FUNCTION_BLOCK ABSTRACT FB_ESSMonitoringBase
VAR_INPUT
    nEcMasterNetId: T_AmsNetId;
    iSafetyProvider: I_SafetyProvider;
END_VAR
VAR_OUTPUT
    aErrorID: ARRAY [1..nMAX_ALARMS] OF INT;
    aErrorMsg: ARRAY [1..nMAX_ALARMS] OF STRING;
    nEcMasterFramesLost: UDINT;
    nCPULoad: UDINT;
    fCycleExecTime_ms: REAL;
    nAlarmGrpBitNumber: UDINT;
END_VAR
VAR
    _bErrorAcknowledgeButton: BOOL;
    _bErrorAcknowledgeLED: BOOL;
    _bStatusLED: BOOL;
    _bEStopLED: BOOL;
    _bErrorLED: BOOL;
    _bEStopReleased: BOOL;
    _nEcMasterDevState: UINT;

    aAlarmList: ARRAY [1..nMAX_ALARMS] OF ST_MonitoringAlarm := [
(*[1]*)(nErrorID:=241, sErrorMsg:='The DC OK Status from PS 24V-1 is OFF.', eStatusLED:=E_MonitorLed.eFast, eErrorLED:=E_MonitorLed.eSteady),
(*[2]*)(nErrorID:=242, sErrorMsg:='The DC OK Status from PS 24V-2 is OFF.', eStatusLED:=E_MonitorLed.eFast, eErrorLED:=E_MonitorLed.eSteady),
(*[3]*)(nErrorID:=243, sErrorMsg:='The DC OK Status from PS 24V-3 is OFF.', eStatusLED:=E_MonitorLed.eFast, eErrorLED:=E_MonitorLed.eSteady),
(*[4]*)(nErrorID:=481, sErrorMsg:='The DC OK Status from PS 48V-1 is OFF.', eStatusLED:=E_MonitorLed.eFast, eErrorLED:=E_MonitorLed.eSteady),
(*[5]*)(nErrorID:=482, sErrorMsg:='The DC OK Status from PS 48V-2 is OFF.', eStatusLED:=E_MonitorLed.eFast, eErrorLED:=E_MonitorLed.eSteady),
(*[6]*)(nErrorID:=483, sErrorMsg:='The DC OK Status from PS 48V-3 is OFF.', eStatusLED:=E_MonitorLed.eFast, eErrorLED:=E_MonitorLed.eSteady),
(*[7]*)(nErrorID:=484, sErrorMsg:='The DC OK Status from PS 48V-4 is OFF.', eStatusLED:=E_MonitorLed.eFast, eErrorLED:=E_MonitorLed.eSteady),
(*[8]*)(nErrorID:=11, sErrorMsg:='MCB Fan OK status is OFF', eStatusLED:=E_MonitorLed.eFast, eErrorLED:=E_MonitorLed.eSteady),
(*[9]*)(nErrorID:=12, sErrorMsg:='SPD OK status is OFF', eStatusLED:=E_MonitorLed.eFast, eErrorLED:=E_MonitorLed.eSteady),
(*[10]*)(nErrorID:=13, sErrorMsg:='Cabinet door Opened', eStatusLED:=E_MonitorLed.eSteady, eErrorLED:=E_MonitorLed.eSteady, bLedAutoReset:=TRUE),
(*[11]*)(nErrorID:=301, sErrorMsg:='Fuse 1 tripped', eStatusLED:=E_MonitorLed.eUndefined, eErrorLED:=E_MonitorLed.eUndefined),
(*[12]*)(nErrorID:=302, sErrorMsg:='Fuse 2 tripped', eStatusLED:=E_MonitorLed.eSlow, eErrorLED:=E_MonitorLed.eSteady),
(*[13]*)(nErrorID:=303, sErrorMsg:='Fuse 3 tripped', eStatusLED:=E_MonitorLed.eSlow, eErrorLED:=E_MonitorLed.eSteady),
(*[14]*)(nErrorID:=304, sErrorMsg:='Fuse 4 tripped', eStatusLED:=E_MonitorLed.eSlow, eErrorLED:=E_MonitorLed.eUndefined),
(*[15]*)(nErrorID:=305, sErrorMsg:='Fuse 5 tripped', eStatusLED:=E_MonitorLed.eSlow, eErrorLED:=E_MonitorLed.eUndefined),
(*[16]*)(nErrorID:=306, sErrorMsg:='Fuse 6 tripped', eStatusLED:=E_MonitorLed.eSlow, eErrorLED:=E_MonitorLed.eUndefined),
(*[17]*)(nErrorID:=307, sErrorMsg:='Fuse 7 tripped', eStatusLED:=E_MonitorLed.eSlow, eErrorLED:=E_MonitorLed.eUndefined),
(*[18]*)(nErrorID:=308, sErrorMsg:='Fuse 8 tripped', eStatusLED:=E_MonitorLed.eSlow, eErrorLED:=E_MonitorLed.eUndefined),
(*[19]*)(nErrorID:=501, sErrorMsg:='E-Stop active', eStatusLED:=E_MonitorLed.eSteady, eErrorLED:=E_MonitorLed.eUndefined, eEStopLED:=E_MonitorLed.eSteady, bLedAutoReset:=TRUE),
(*[20]*)(nErrorID:=14, sErrorMsg:='Temperature 1 too high', eStatusLED:=E_MonitorLed.eUndefined, eErrorLED:=E_MonitorLed.eSteady),
(*[21]*)(nErrorID:=15, sErrorMsg:='Temperature 2 too high', eStatusLED:=E_MonitorLed.eUndefined, eErrorLED:=E_MonitorLed.eSteady),
(*[22]*)(nErrorID:=16, sErrorMsg:='Temperature 3 too high', eStatusLED:=E_MonitorLed.eUndefined, eErrorLED:=E_MonitorLed.eSteady),
(*[23]*)(nErrorID:=17, sErrorMsg:='Temperature 4 too high', eStatusLED:=E_MonitorLed.eUndefined, eErrorLED:=E_MonitorLed.eSteady),
(*[24]*)(nErrorID:=101, sErrorMsg:='EtherCAT Master is not ok', eStatusLED:=E_MonitorLed.eSteady, eErrorLED:=E_MonitorLed.eUndefined),
(*[25]*)(nErrorID:=102, sErrorMsg:='EtherCAT slave(s) not in OP state', eStatusLED:=E_MonitorLed.eSteady, eErrorLED:=E_MonitorLed.eSteady),
(*[26]*)(nErrorID:=103, sErrorMsg:='EtherCAT slave(s) link fault', eStatusLED:=E_MonitorLed.eSteady, eErrorLED:=E_MonitorLed.eSteady),
(*[27]*)(nErrorID:=104, sErrorMsg:='Overflow in PLC cycle time', eStatusLED:=E_MonitorLed.eSteady, eErrorLED:=E_MonitorLed.eUndefined),
(*[28]*)(nErrorID:=105, sErrorMsg:='CPU Load High', eStatusLED:=E_MonitorLed.eSteady, eErrorLED:=E_MonitorLed.eUndefined),
(*[29]*)(nErrorID:=18, sErrorMsg:='MCB Piezo Controller Off', eStatusLED:=E_MonitorLed.eFast, eErrorLED:=E_MonitorLed.eSteady),
(*[30]*)(nErrorID:=19, sErrorMsg:='MCB VFD Off', eStatusLED:=E_MonitorLed.eFast, eErrorLED:=E_MonitorLed.eSteady),
(*[31]*)(nErrorID:=601, sErrorMsg:='Shutter OP Fuse 1 tripped', eStatusLED:=E_MonitorLed.eUndefined, eErrorLED:=E_MonitorLed.eUndefined, bLedAutoReset:=TRUE),
(*[32]*)(nErrorID:=602, sErrorMsg:='Shutter OP Fuse 2 tripped', eStatusLED:=E_MonitorLed.eUndefined, eErrorLED:=E_MonitorLed.eUndefined, bLedAutoReset:=TRUE),
(*[33]*)(nErrorID:=603, sErrorMsg:='Shutter OP DC OK Status from PS 24V is OFF.', eStatusLED:=E_MonitorLed.eFast, eErrorLED:=E_MonitorLed.eSteady, bLedAutoReset:=TRUE),
(*[34]*)(nErrorID:=604, sErrorMsg:='Shutter OP SPD OK status is OFF', eStatusLED:=E_MonitorLed.eFast, eErrorLED:=E_MonitorLed.eSteady, bLedAutoReset:=TRUE),
(*[35]*)(nErrorID:=701, sErrorMsg:='EC Nodebox Fuse 1 tripped', eStatusLED:=E_MonitorLed.eUndefined, eErrorLED:=E_MonitorLed.eUndefined, bLedAutoReset:=TRUE),
(*[36]*)(nErrorID:=702, sErrorMsg:='EC Nodebox Fuse 2 tripped', eStatusLED:=E_MonitorLed.eUndefined, eErrorLED:=E_MonitorLed.eUndefined, bLedAutoReset:=TRUE),
(*[37]*)(nErrorID:=703, sErrorMsg:='EC Nodebox DC OK Status from PS 24V-1 is OFF.', eStatusLED:=E_MonitorLed.eFast, eErrorLED:=E_MonitorLed.eSteady, bLedAutoReset:=TRUE),
(*[38]*)(nErrorID:=704, sErrorMsg:='EC Nodebox DC OK Status from PS 24V-2 is OFF.', eStatusLED:=E_MonitorLed.eFast, eErrorLED:=E_MonitorLed.eSteady, bLedAutoReset:=TRUE),
(*[39]*)(nErrorID:=705, sErrorMsg:='EC Nodebox SPD OK status is OFF', eStatusLED:=E_MonitorLed.eFast, eErrorLED:=E_MonitorLed.eSteady, bLedAutoReset:=TRUE)];


    aTempErrorID: ARRAY [1..nMAX_ALARMS] OF INT;
    aTempErrorMsg: ARRAY [1..nMAX_ALARMS] OF STRING;

    nAlarmCnt: INT;
    nAlarmBitNumber: UDINT;

    bCPUOverloaded: BOOL;
    bEcMasterError: BOOL;
    bSlaveStateNotOP: BOOL;
    bSlaveLinkError: BOOL;
    aExtraMessage: ARRAY[1..nMAX_ALARMS] OF STRING := [nMAX_ALARMS('')];
    bCycleTimeExceeded: BOOL;

    //Ethercat master device state
    bEcLinkError: BOOL;
    bEcIOlocked: BOOL;
    bEcLinkErrorRedundancyAdapter: BOOL;
    bEcMissingFrame: BOOL;
    bEcOutofSendResources: BOOL;
    bEcWatchdogTriggered: BOOL;
    bEcEthernetDriverNotFound: BOOL;
    bEcIOresetActive: BOOL;
    bEcSlaveINIT: BOOL;
    bEcSlavePreOP: BOOL;
    bEcSlaveSafeOP: BOOL;
    bEcSlaveError: BOOL;
    bEcDCnotInSync: BOOL;

    //Data from the safety controller
    _EStopReleased: BOOL;
    _STOReleased: BOOL;

    fbAcknowledgeButtonTrig: R_TRIG;
END_VAR

VAR CONSTANT
    tNEW_MESSAGE_TIMEOUT: TIME := T#300S;
    nMAX_ALARMS: UINT := 50;
    nMAX_EC_SLAVES: INT := 255;
    nMAX_TEMP: INT := 10000;
    nSLAVE_NOT_OP_STATE_ENTRY: UDINT := 28;
    nSLAVE_LINK_ERROR_ENTRY: UDINT := 29;
END_VAR

mMonitorAlarms();
mMonitorCPU();
mMonitorEtherCAT();
mLink();

PROPERTY PROTECTED AcknowledgeButton : BOOL
SET
_bErrorAcknowledgeButton := AcknowledgeButton;
END_SET
END_PROPERTY

PROPERTY AcknowledgeLED : BOOL
GET
AcknowledgeLED := _bErrorAcknowledgeLED;
END_GET
END_PROPERTY

PROPERTY EcMasterDevState : UINT
SET
_nEcMasterDevState := EcMasterDevState;
END_SET
END_PROPERTY

PROPERTY PROTECTED ErrorLED : BOOL
GET
ErrorLED := _bErrorLED;
END_GET
END_PROPERTY

PROPERTY PROTECTED EStopLED : BOOL
GET
EStopLED := _bEStopLED;
END_GET
END_PROPERTY

PROPERTY PUBLIC EStopReleased : BOOL
GET
EStopReleased := _bEStopReleased;
END_GET
SET
_bEStopReleased := EStopReleased;
END_SET
END_PROPERTY

METHOD FB_init : BOOL
VAR_INPUT
    bInitRetains : BOOL; // if TRUE, the retain variables are initialized (warm start / cold start)
    bInCopyCode : BOOL;  // if TRUE, the instance afterwards gets moved into the copy code (online change)
END_VAR

VAR
    i : UINT := 0;
END_VAR
FOR i := 1 TO THIS^.nMAX_ALARMS DO
    IF THIS^.aAlarmList[i].bLedAutoReset THEN
        THIS^.aAlarmList[i].eErrorAcknowledgeLED := E_MonitorLed.eUndefined;
    ELSE
        THIS^.aAlarmList[i].eErrorAcknowledgeLED := E_MonitorLed.eSteady;
    END_IF
END_FOR
END_METHOD

METHOD mAlarmActive
VAR_INPUT
    i: UINT;
    bUpdatedExtraMessage : BOOL;
END_VAR

VAR_INST
    aFbErrorMessageTimer: ARRAY[1..nMAX_ALARMS] OF TON;
    aStartErrorMsgTimer: ARRAY[1..nMAX_ALARMS] OF BOOL;
    aFbErrorTrig: ARRAY[1..nMAX_ALARMS] OF R_TRIG;
END_VAR
// Update timer and trigger for new log message
aStartErrorMsgTimer[i] :=
    aAlarmList[i].bAlarmActive
    AND NOT aFbErrorMessageTimer[i].Q;
aFbErrorMessageTimer[i](
    IN:=aStartErrorMsgTimer[i],
    PT:=tNEW_MESSAGE_TIMEOUT);
aFbErrorTrig[i](
    CLK:=aStartErrorMsgTimer[i]);

IF NOT aAlarmList[i].bAlarmActive THEN
    RETURN;
END_IF

nAlarmCnt := nAlarmCnt + 1;
aTempErrorID[nAlarmCnt] := aAlarmList[i].nErrorID;
aTempErrorMsg[nAlarmCnt] := CONCAT(aAlarmList[i].sErrorMsg, aExtraMessage[i]);

mPrintErrorMessage(
    bPrintLog:=aFbErrorTrig[i].Q OR bUpdatedExtraMessage,
    sErrorMessage:=aTempErrorMsg[nAlarmCnt],
    nErrorID:=aAlarmList[i].nErrorID,
    nIndex:=i);

// Map nErrorID to nAlarmBitnumber, which later is mapped to output variable nAlarmGrpBitNumber.
CASE aAlarmList[i].nErrorID OF
    241, 242, 243:
    nAlarmBitNumber.0 := TRUE;
    481, 482, 483, 484:
    nAlarmBitNumber.1 := TRUE;
    11:
    nAlarmBitNumber.2 := TRUE;
    12:
    nAlarmBitNumber.3 := TRUE;
    13:
    nAlarmBitNumber.4 := TRUE;
    14,15,16,17:
    nAlarmBitNumber.5 := TRUE;
    301, 302, 303, 304, 305, 306, 307, 308:
    nAlarmBitNumber.6 := TRUE;
    501, 502, 511, 512:
    nAlarmBitNumber.7 := TRUE;
    101:
    nAlarmBitNumber.8 := TRUE;
    102:
    nAlarmBitNumber.9 := TRUE;
    103:
    nAlarmBitNumber.10 := TRUE;
    104, 105:
    nAlarmBitNumber.11 := TRUE;
    18,19:
    nAlarmBitNumber.12 := TRUE;
END_CASE
END_METHOD

METHOD ABSTRACT mLink
END_METHOD

METHOD mMonitorAlarms
VAR
    i: UINT := 0;
    stMonitorLed: ST_MonitoringAlarm;
END_VAR

VAR_INST
    aExtraMessageOld: ARRAY[1..nMAX_ALARMS] OF STRING := [nMAX_ALARMS('')];
    bLedActive: BOOL := FALSE;
    fbFastBlinkOn: TON;
    fbFastBlinkOff: TON;
    fbSlowBlinkOn: TON;
    fbSlowBlinkOff: TON;
END_VAR
fbAcknowledgeButtonTrig(CLK:=_bErrorAcknowledgeButton);
mSetResetAlarmsLeds();

// Reset before loop
nAlarmCnt := 0;
nAlarmBitNumber := 0;
MEMSET(ADR(aTempErrorID), 0, SIZEOF(aTempErrorID));
MEMSET(ADR(aTempErrorMsg), 0, SIZEOF(aTempErrorMsg));
bLedActive := FALSE;

FOR i:=1 TO nMAX_ALARMS DO
    // Handle log prints, alarm bits and prepare alarm LEDs
    mAlarmActive(i:=i, bUpdatedExtraMessage := aExtraMessage[i] <> aExtraMessageOld[i]);

    // Set the alarm LEDs according to first occurrence
    IF NOT bLedActive
        AND aAlarmList[i].bLedActive THEN
        bLedActive := TRUE;
        stMonitorLed.eErrorLED := aAlarmList[i].eErrorLED;
        stMonitorLed.eStatusLED := aAlarmList[i].eStatusLED;
    END_IF

    // If any error exists requiring an acknowledge, highlight Acknowledge LED.
    IF aAlarmList[i].bLedActive AND NOT aAlarmList[i].bLedAutoReset THEN
        stMonitorLed.eErrorAcknowledgeLED := aAlarmList[i].eErrorAcknowledgeLED;
    END_IF
END_FOR

// Save last messages for next iteration
aExtraMessageOld := aExtraMessage;

// Copy to output variables
aErrorID := aTempErrorID;
aErrorMsg := aTempErrorMsg;
nAlarmGrpBitNumber := nAlarmBitNumber;

// Handle LED blinking
fbFastBlinkOn(IN:=NOT fbFastBlinkOff.Q, PT:=T#250MS);
fbFastBlinkOff(IN:=fbFastBlinkOn.Q, PT:=T#250MS);

fbSlowBlinkOn(IN:=NOT fbSlowBlinkOff.Q, PT:=T#750MS);
fbSlowBlinkOff(IN:=fbSlowBlinkOn.Q, PT:=T#750MS);

_bErrorLED :=
    (stMonitorLed.eErrorLED = E_MonitorLed.eSteady)
    OR (stMonitorLed.eErrorLED = E_MonitorLed.eFast AND fbFastBlinkOn.Q)
    OR (stMonitorLed.eErrorLED = E_MonitorLed.eSlow AND fbSlowBlinkOn.Q);
_bStatusLED :=
    (stMonitorLed.eStatusLED = E_MonitorLed.eSteady)
    OR (stMonitorLed.eStatusLED = E_MonitorLed.eFast AND fbFastBlinkOn.Q)
    OR (stMonitorLed.eStatusLED = E_MonitorLed.eSlow AND fbSlowBlinkOn.Q);
_bErrorAcknowledgeLED :=
    (stMonitorLed.eErrorAcknowledgeLED = E_MonitorLed.eSteady)
    OR (stMonitorLed.eErrorAcknowledgeLED = E_MonitorLed.eFast AND fbFastBlinkOn.Q)
    OR (stMonitorLed.eErrorAcknowledgeLED = E_MonitorLed.eSlow AND fbSlowBlinkOn.Q);
_bEStopLED := NOT _bEStopReleased;
END_METHOD

METHOD mMonitorCPU

VAR_INST
    fbMonitorCPU: TC_CpuUsage;
    fbUpdateCPULoadTON: TON;
    fMaxCPULoad: USINT := 85;
END_VAR
//Cpu Monitor
fbUpdateCPULoadTON(IN:=NOT fbUpdateCPULoadTON.q , PT:=T#100MS , Q=> , ET=> );
fbMonitorCPU(START:=fbUpdateCPULoadTON.q, TMOUT:= T#5S);

bCPUOverloaded := fbMonitorCPU.USAGE > fMaxCPULoad;
nCPULoad := fbMonitorCPU.USAGE;

fCycleExecTime_ms := UDINT_TO_REAL(_TaskInfo[fbGetCurTaskIndex.index].LastExecTime) / 10000;
bCycleTimeExceeded := _TaskInfo[fbGetCurTaskIndex.index].CycleTimeExceeded;
END_METHOD

METHOD mMonitorEtherCAT
VAR
    i: UINT := 0;
END_VAR

VAR_INST
    fbGetEcSlaveStates: FB_EcGetAllSlaveStates;
    stSlaveState: ARRAY[0..nMAX_EC_SLAVES] OF ST_EcSlaveState;
    nActualEcSlaves: UINT := 0;
    fbGetEcConfSlaves: FB_EcGetConfSlaves;
    aSlaveConfigBuffer1: ARRAY[1..EC_MAX_SLAVES] OF ST_EcSlaveConfigData; //Buffer 1 for EtherCAT Slave Config Data
    aSlaveConfigBuffer2: ARRAY[1..EC_MAX_SLAVES] OF ST_EcSlaveConfigData; //Buffer 2 for EtherCAT Slave Config Data
    pWriteSlaveConfigBuffer: POINTER TO ARRAY[1..EC_MAX_SLAVES] OF ST_EcSlaveConfigData; //Pointer to the buffer with write access
    pReadSlaveConfigBuffer: POINTER TO ARRAY[1..EC_MAX_SLAVES] OF ST_EcSlaveConfigData; //Pointer to the buffer with read access
    fbGetEcMasterFrames: FB_EcMasterFrameStatistic;
    tonAutoResetError: TON;
    bFirstReadSlaveConfigDone: BOOL := FALSE;
    bErrorZeroEcSlavesFound: BOOL := FALSE;
    bInit: BOOL := TRUE;
END_VAR
VAR CONSTANT
    tAUTO_RESET: TIME := T#3S;
END_VAR
IF bInit THEN
    bInit := FALSE;
    pWriteSlaveConfigBuffer := ADR(aSlaveConfigBuffer1);
    pReadSlaveConfigBuffer := ADR(aSlaveConfigBuffer2);
END_IF

tonAutoResetError(
    PT := tAUTO_RESET,
    IN := NOT tonAutoResetError.Q
        AND (fbGetEcMasterFrames.bError
        OR fbGetEcConfSlaves.bError
        OR fbGetEcSlaveStates.bError));

//Read the frame statistics of the EtherCAT master.
fbGetEcMasterFrames(
    sNetId := nEcMasterNetId,
    bExecute := NOT (fbGetEcMasterFrames.bBusy
        OR fbGetEcMasterFrames.bError)
        OR tonAutoResetError.Q);
nEcMasterFramesLost := fbGetEcMasterFrames.nLostFrames;

//Read a list of configured slaves from the EtherCAT master object directory.
fbGetEcConfSlaves(
    sNetId := nEcMasterNetId,
    pArrEcConfSlaveInfo := pWriteSlaveConfigBuffer,
    cbBufLen := SIZEOF(pWriteSlaveConfigBuffer^),
    bExecute := NOT (fbGetEcConfSlaves.bBusy
        OR fbGetEcConfSlaves.bError)
        OR tonAutoResetError.Q);

//Swap buffer if read out is sucessfully finishes
IF NOT (fbGetEcConfSlaves.bBusy
    OR fbGetEcConfSlaves.bError
    OR fbGetEcConfSlaves.nSlaves = 0)
THEN
    bFirstReadSlaveConfigDone := TRUE;
    IF pWriteSlaveConfigBuffer = ADR(aSlaveConfigBuffer1) THEN
        pWriteSlaveConfigBuffer := ADR(aSlaveConfigBuffer2);
        pReadSlaveConfigBuffer := ADR(aSlaveConfigBuffer1);
    ELSE
        pWriteSlaveConfigBuffer := ADR(aSlaveConfigBuffer1);
        pReadSlaveConfigBuffer := ADR(aSlaveConfigBuffer2);
    END_IF
END_IF

//Get EtherCAT status and the Link status of all the slaves connected to the master.
fbGetEcSlaveStates(
    sNetId := nEcMasterNetId,
    pStateBuf := ADR(stSlaveState),
    cbBufLen := SIZEOF(stSlaveState),
    //fbGetEcSlaveStates never goes bBusy (finishes same cycle as bExecute)
    //Starts on bExecute of fbGetEcConfSlaves instead
    bExecute := (fbGetEcConfSlaves.bExecute
        AND NOT fbGetEcSlaveStates.bError)
        OR tonAutoResetError.Q);
nActualEcSlaves := fbGetEcSlaveStates.nSlaves;

//Check ethercat master device state
bEcLinkError := _nEcMasterDevState.0;
bEcIOlocked := _nEcMasterDevState.1;
bEcLinkErrorRedundancyAdapter := _nEcMasterDevState.2;
bEcMissingFrame := _nEcMasterDevState.3;
bEcOutofSendResources := _nEcMasterDevState.4;
bEcWatchdogTriggered := _nEcMasterDevState.5;
bEcEthernetDriverNotFound := _nEcMasterDevState.6;
bEcIOresetActive := _nEcMasterDevState.7;
bEcSlaveINIT := _nEcMasterDevState.8;
bEcSlavePreOP := _nEcMasterDevState.9;
bEcSlaveSafeOP := _nEcMasterDevState.10;
bEcSlaveError := _nEcMasterDevState.11;
bEcDCnotInSync := _nEcMasterDevState.12;

bEcMasterError := _nEcMasterDevState > 0;

//After startup reset variables before loop
bSlaveStateNotOP := FALSE;
bSlaveLinkError := FALSE;
aExtraMessage[nSLAVE_NOT_OP_STATE_ENTRY] := ', Slave Id #: ';
aExtraMessage[nSLAVE_LINK_ERROR_ENTRY] := ', Slave Id #: ';

IF nActualEcSlaves = 0 THEN
    IF NOT bErrorZeroEcSlavesFound THEN
        bErrorZeroEcSlavesFound := TRUE;
        ADSLOGSTR(
            msgCtrlMask := ADSLOG_MSGTYPE_ERROR,
            msgFmtStr := 'FB_ESSMonitoringBase Error: %s',
            strArg := '0 EtherCAT Slaves found, check correct AmsNetId in CabinetMonitoring');
    END_IF
    bSlaveLinkError := TRUE;
    aExtraMessage[nSLAVE_LINK_ERROR_ENTRY] := ', 0 EtherCAT Slaves found';
    RETURN;
END_IF
bErrorZeroEcSlavesFound := FALSE;

IF NOT bFirstReadSlaveConfigDone THEN
    RETURN;
END_IF

FOR i:=0 TO nActualEcSlaves-1 DO
    IF stSlaveState[i].linkState <> EC_LINK_STATE_OK  THEN
        aExtraMessage[nSLAVE_LINK_ERROR_ENTRY] :=
            CONCAT(STR1:=aExtraMessage[nSLAVE_LINK_ERROR_ENTRY], STR2:=UINT_TO_STRING(i+1));
        IF NOT bSlaveLinkError THEN
            aExtraMessage[nSLAVE_LINK_ERROR_ENTRY] :=
                CONCAT(STR1:=aExtraMessage[nSLAVE_LINK_ERROR_ENTRY], STR2:=CONCAT('-', LEFT(pReadSlaveConfigBuffer^[i+1].sName, FIND(pReadSlaveConfigBuffer^[i+1].sName,' (')-1)));
        END_IF
        aExtraMessage[nSLAVE_LINK_ERROR_ENTRY] :=
            CONCAT(STR1:=aExtraMessage[nSLAVE_LINK_ERROR_ENTRY], STR2:=', ');
        bSlaveLinkError := TRUE;
        // Do not print slave numbers for deviceState if already printed for linkState
        CONTINUE;
    END_IF

    IF stSlaveState[i].deviceState <> EC_DEVICE_STATE_OP THEN
        aExtraMessage[nSLAVE_NOT_OP_STATE_ENTRY] :=
            CONCAT(STR1:=aExtraMessage[nSLAVE_NOT_OP_STATE_ENTRY], STR2:= UINT_TO_STRING(i+1));
        IF NOT bSlaveStateNotOP THEN
            aExtraMessage[nSLAVE_NOT_OP_STATE_ENTRY] :=
                CONCAT(STR1:=aExtraMessage[nSLAVE_NOT_OP_STATE_ENTRY], STR2:=CONCAT('-', LEFT(pReadSlaveConfigBuffer^[i+1].sName, FIND(pReadSlaveConfigBuffer^[i+1].sName,' (')-1)));
        END_IF
        aExtraMessage[nSLAVE_NOT_OP_STATE_ENTRY] :=
            CONCAT(STR1:=aExtraMessage[nSLAVE_NOT_OP_STATE_ENTRY], STR2:=', ');
        bSlaveStateNotOP := TRUE;
    END_IF
END_FOR
END_METHOD

METHOD mPrintErrorMessage
VAR_INPUT
    bPrintLog : BOOL;
    sErrorMessage: STRING;
    nErrorID: INT;
    nIndex: UINT;
END_VAR
VAR
    sErrorId: STRING;
END_VAR
IF NOT bPrintLog THEN
    RETURN;
END_IF

sErrorId := CONCAT(STR1:='ErrorID: ', STR2:=INT_TO_STRING(nErrorID));
sErrorId := CONCAT(STR1:=sErrorId, STR2:='. %s');

ADSLOGSTR(
    msgCtrlMask:=ADSLOG_MSGTYPE_ERROR,
    msgFmtStr:=sErrorId,
    strArg:=sErrorMessage);
END_METHOD

METHOD mSetReset
VAR_INPUT
    bOk: BOOL;
END_VAR

VAR_IN_OUT
    stAlarmList: ST_MonitoringAlarm;
END_VAR
IF NOT bOk THEN
    stAlarmList.bAlarmActive := TRUE;
    stAlarmList.bLedActive := TRUE;
    RETURN;
END_IF

stAlarmList.bAlarmActive := FALSE;

IF stAlarmList.bLedAutoReset OR fbAcknowledgeButtonTrig.Q THEN
    stAlarmList.bLedActive := FALSE;
END_IF
END_METHOD

METHOD ABSTRACT mSetResetAlarmsLeds
END_METHOD

PROPERTY PROTECTED StatusLED : BOOL
GET
StatusLED := _bStatusLED;
END_GET
END_PROPERTY

END_FUNCTION_BLOCK

(* stored: Version 1.1.0.1
   POU FB_ESSMonitoringBase: Id {16375c53-a76d-0f86-34ec-9cedc05223d1}, SpecialFunc None
   Property AcknowledgeButton: Id {4553ddaa-9a47-067f-1824-16747e3b18bb}
   Set Set: Id {097bd8e4-8f42-0d2f-3b2d-68c813444beb}
   Property AcknowledgeLED: Id {87e182de-d7eb-0e63-0a1a-4287ee4dac3d}
   Get Get: Id {c85992ab-d415-0e8f-2295-5c0c5b4bcb43}
   Property EcMasterDevState: Id {4d86de19-f4c1-0929-075b-548e5f42ca15}
   Set Set: Id {17101c7e-75b1-0240-27ab-ffc2d1577fcb}
   Property ErrorLED: Id {7eb12b12-2c1a-030f-02c0-dc876b161c7d}
   Get Get: Id {dee2b4e1-cf32-02a5-164a-d408751a1e36}
   Property EStopLED: Id {11c0d295-1ba3-0cb3-34ae-5cedaebe894d}
   Get Get: Id {c6083b86-6c45-076c-267f-649012ee9fb9}
   Property EStopReleased: Id {0f76b944-cd05-0d53-20d1-3839916d7d3a}
   Get Get: Id {a27c5f82-1830-0be3-27f0-6e9ced4ccd5e}
   Set Set: Id {2d659b6b-6763-0d53-355a-5af1c0fcb381}
   Method FB_init: Id {fbc6fe99-d298-01aa-2f2e-75ad59229db1}
   Method mAlarmActive: Id {aff05498-00f1-0703-1f58-de4c9fc3cb2d}
   Method mLink: Id {92e02a6e-69e5-0850-2551-9162736c466e}
   Method mMonitorAlarms: Id {542f94fc-2447-0df7-2067-48b1bdc9c1ba}
   Method mMonitorCPU: Id {a61c27e8-4c84-0867-118e-ec0a5a4d454e}
   Method mMonitorEtherCAT: Id {27ca7522-14a9-0d7c-33ae-0dd2d861dfe1}
   Method mPrintErrorMessage: Id {3e321397-22af-4d7e-a9bd-c132b0a3b842}
   Method mSetReset: Id {bc20beb2-4ad1-01ee-3c55-7ebdd0373966}
   Method mSetResetAlarmsLeds: Id {b9cbdba3-25a5-0522-2be9-bdaa3a3049b0}
   Property StatusLED: Id {aae8b4d5-2209-0213-0845-6c75706f0ec1}
   Get Get: Id {771086b7-4d2a-0e03-15a1-c2c5934c123b} *)
